(* IEC 61131-3 sources: Industry-PLC-LLM/data/PLCBEAD_repo/PLCBEAD_PLCEmbed-main/PLC-BEAD/Source/GEB/Network_TN_SEND_ROWS, 1 file *)

(* ---- TN_SEND_ROWS.ST ---- *)
TYPE
  oscat_IP_FIFO128_DATA  : ARRAY [1..128] OF BYTE;
  oscat_Mailbox  : ARRAY [1..16] OF BYTE;

  oscat_IP_FIFO_DATA :
  STRUCT
    X       : oscat_IP_FIFO128_DATA; (* IP_ID FIFO Speicher          *)
    Y       : oscat_IP_FIFO128_DATA; (* IP_ID Z�hler                 *)
    ID      : BYTE;                  (* h�chste vergabene id         *)
    MAX_ID  : BYTE;                  (* maximal Anmeldungen pro ID   *)
    INIT    : BOOL;                  (* Initialisierung durchgef�hrt *)
    EMPTY   : BOOL;                  (* FIFO leer                    *)
    FULL    : BOOL;                  (* FIFO voll                    *)
    TOP     : INT;                   (* maximale anzahl IN FIFO      *)
    NW      : INT;                   (* Schreibzeiger                *)
    NR      : INT;                   (* Lesezeiger                   *)
  END_STRUCT;

  oscat_IP_C:
  STRUCT
    C_MODE:			BYTE;          		(*W Mode: TCP/UCP AKTIV/PASSIV                               *)
    C_PORT:         WORD;          		(*W Portnummer                                               *)
    C_IP:           DWORD;         		(*W IP-ADRESSe gepackt wwxxyyzz = www.xxx.yyy.zzz            *)
    C_STATE:        BYTE;          		(*R VerbindungsSTATUS ON/OFF + Flanke ON/OFF                 *)
    C_ENABLE:       BOOL;          		(*W Freigabe f�r Connect                                     *)
    R_OBSERVE:      BOOL;          		(*W Empfang ueberwachen                                      *)
    TIME_RESET:     BOOL;          		(*W Alle Timer ruecksetzen                                   *)
    ERROR:          DWORD;         		(*R vvwwxxyy (vv = CON_ERROR, ww = SEN_ERROR, xx = REC_ERROR *)
    FIFO:           oscat_IP_FIFO_DATA; (*I IP FIFO Struktur                                         *)
    MAILBOX:		oscat_Mailbox;		(*I Mailbox: Datenbereich f�r Bausteindatenaustausch         *)
    END_STRUCT;
END_TYPE

TYPE

  oscat_NW_BUF_LONG  : ARRAY [0..4095] OF BYTE;

  oscat_NETWORK_BUFFER :
  STRUCT
    SIZE   : UINT;
    BUFFER : oscat_NW_BUF_LONG;
  END_STRUCT;

END_TYPE

TYPE

  bya_TN_CHAR:       	ARRAY [0..1919] OF BYTE;
  bya_TN_BACKUP:     	ARRAY [0..1919] OF BYTE;
  bya_TN_COLOR:      	ARRAY [0..1919] OF BYTE;
  bya_TN_Line_Update:	ARRAY [0..23]   OF BOOL;

  us_TN_SCREEN :
  STRUCT
    bya_CHAR:			bya_TN_CHAR;
    bya_COLOR:			bya_TN_COLOR;
    bya_BACKUP:			bya_TN_BACKUP;
    bya_Line_Update:	bya_TN_Line_Update;

    by_Input_Exten_Code:    BYTE;
    by_Input_ASCII_Code:    BYTE;
    bo_Input_ASCII_IsNum:   BOOL;
    in_Page_Number:        	INT;                (* aktive Seiten-Nr.              *)
    in_Cursor_X:           	INT;                (* Cursor X-POSition              *)
    in_Cursor_Y:           	INT;                (* Cursor Y-POSition              *)
    in_EOS_Offset:         	INT;                (* End of String Offset           *)
    by_Clear_Screen_Attr:  	BYTE;               (* Clear-Screen Attr              *)
    bo_Clear_Screen:       	BOOL;               (* Clear-Screen ausl�sen          *)
    bo_Modal_Dialog:       	BOOL;               (* Modaler Dialog ist aktiv       *)
    bo_Menue_Bar_Dialog:   	BOOL;               (* Menue Dialog ist aktiv         *)

  END_STRUCT;
END_TYPE

FUNCTION INT_TO_BCDC:BYTE

	VAR_INPUT
		IN :	INT;
	END_VAR

	INT_TO_BCDC := SHL(INT_TO_BYTE(IN / INT#10),4) OR INT_TO_BYTE(IN MOD INT#10);

END_FUNCTION

FUNCTION_BLOCK TN_SEND_ROWS_Block

  VAR_IN_OUT
    IP_C :	oscat_IP_C;
    S_BUF :	oscat_NETWORK_BUFFER;
    Xus_TN_SCREEN :	us_TN_SCREEN;
  END_VAR

  VAR_INPUT
    S_BUF_SIZE :	INT;
  END_VAR

  VAR
    in_Line_Count :	INT;
    in_Col_Count :	INT;
    in_Last_Row_Index :	INT;
    bo_Break_Loop :	BOOL;
    in_Row_Count :	INT;
    in_Offset :	INT;
    in_Write_Index :	INT;
    in_Write_Index_Backup :	INT;
    by_Cur_Color :	BYTE;
    by_last_Color :	BYTE;
    in_Write_STOP :	INT;
  END_VAR

  IF (IP_C.C_STATE < BYTE#127 OR S_BUF.SIZE > UINT#0) THEN
    RETURN;
  END_IF;

  in_Write_Index := UINT_TO_INT(S_BUF.SIZE) - 1;

  in_Write_Index_Backup := in_Write_Index;

  IF (IP_C.C_STATE = BYTE#254) OR (Xus_TN_SCREEN.bo_Clear_Screen) THEN

    Xus_TN_SCREEN.bo_Clear_Screen := FALSE;

    FOR in_Line_Count := INT#00 TO INT#23 DO
      Xus_TN_SCREEN.bya_Line_Update[in_Line_Count] := TRUE;
    END_FOR;

    in_Write_Index := in_Write_Index + INT#1;
    S_BUF.BUFFER[in_Write_Index] := BYTE#16#1B;
    in_Write_Index := in_Write_Index + INT#1;
    S_BUF.BUFFER[in_Write_Index] := BYTE#16#5B;
    in_Write_Index := in_Write_Index + INT#1;
    S_BUF.BUFFER[in_Write_Index] := BYTE#16#30;
    in_Write_Index := in_Write_Index + INT#1;
    S_BUF.BUFFER[in_Write_Index] := BYTE#16#3B;
    in_Write_Index := in_Write_Index + INT#1;
    S_BUF.BUFFER[in_Write_Index] := BYTE#16#33;

    in_Write_Index := in_Write_Index + INT#1;
    S_BUF.BUFFER[in_Write_Index] := (SHR(Xus_TN_SCREEN.by_Clear_Screen_Attr,4) OR BYTE#16#30);

    in_Write_Index := in_Write_Index + INT#1;
    S_BUF.BUFFER[in_Write_Index] := BYTE#16#3B;
    in_Write_Index := in_Write_Index + INT#1;
    S_BUF.BUFFER[in_Write_Index] := BYTE#16#34;

    in_Write_Index := in_Write_Index + INT#1;
    S_BUF.BUFFER[in_Write_Index] := ((Xus_TN_SCREEN.by_Clear_Screen_Attr AND BYTE#16#07) OR BYTE#16#30);

    in_Write_Index := in_Write_Index + INT#1;
    S_BUF.BUFFER[in_Write_Index] := BYTE#16#6D;

    in_Write_Index := in_Write_Index + INT#1;
    S_BUF.BUFFER[in_Write_Index] := BYTE#16#1B;
    in_Write_Index := in_Write_Index + INT#1;
    S_BUF.BUFFER[in_Write_Index] := BYTE#16#5B;
    in_Write_Index := in_Write_Index + INT#1;
    S_BUF.BUFFER[in_Write_Index] := BYTE#16#32;
    in_Write_Index := in_Write_Index + INT#1;
    S_BUF.BUFFER[in_Write_Index] := BYTE#16#4A;

    in_Write_Index := in_Write_Index + INT#1;
    S_BUF.BUFFER[in_Write_Index] := BYTE#16#1B;
    in_Write_Index := in_Write_Index + INT#1;
    S_BUF.BUFFER[in_Write_Index] := BYTE#16#5B;
    in_Write_Index := in_Write_Index + INT#1;
    S_BUF.BUFFER[in_Write_Index] := BYTE#16#3F;
    in_Write_Index := in_Write_Index + INT#1;
    S_BUF.BUFFER[in_Write_Index] := BYTE#16#37;
    in_Write_Index := in_Write_Index + INT#1;
    S_BUF.BUFFER[in_Write_Index] := BYTE#16#6C;

  END_IF;

  in_Last_Row_Index := INT#0;
  bo_Break_Loop := FALSE;
  in_Write_STOP := S_BUF_SIZE-20;

  FOR in_Line_Count := 0 TO 23 DO

    in_Offset := in_Row_Count * INT#80;

    IF (Xus_TN_SCREEN.bya_Line_Update[in_Row_Count] = TRUE) THEN

      in_Write_Index := in_Write_Index + INT#1;
      S_BUF.BUFFER[in_Write_Index] := BYTE#16#1B;
      in_Write_Index := in_Write_Index + INT#1;
      S_BUF.BUFFER[in_Write_Index] := BYTE#16#5B;

      in_Write_Index := in_Write_Index + INT#1;
      S_BUF.BUFFER[in_Write_Index] :=
        SHR(INT_TO_BCDC(in_Row_Count + INT#1),INT#4) OR BYTE#16#30;

      in_Write_Index := in_Write_Index + INT#1;
      S_BUF.BUFFER[in_Write_Index] :=
        (INT_TO_BCDC(in_Row_Count + INT#1) AND BYTE#16#0F) OR BYTE#16#30;

      in_Write_Index := in_Write_Index + INT#1;
      S_BUF.BUFFER[in_Write_Index] := BYTE#16#3B;
      in_Write_Index := in_Write_Index + INT#1;
      S_BUF.BUFFER[in_Write_Index] := BYTE#16#31;
      in_Write_Index := in_Write_Index + INT#1;
      S_BUF.BUFFER[in_Write_Index] := BYTE#16#48;

      FOR in_Col_Count := 0 TO 79 DO

        by_Cur_Color := Xus_TN_SCREEN.bya_COLOR[in_Offset];
        IF (by_Cur_Color <> by_last_Color) OR (in_Col_Count = INT#00) THEN

          in_Write_Index := in_Write_Index + INT#1;
          S_BUF.BUFFER[in_Write_Index] := BYTE#16#1B;

          in_Write_Index := in_Write_Index + INT#1;
          S_BUF.BUFFER[in_Write_Index] := BYTE#16#5B;

          IF  (((by_Cur_Color AND BYTE#2#10001000) XOR (by_last_Color AND BYTE#2#10001000)) <> BYTE#00) OR (in_Col_Count = 0) THEN

            in_Write_Index := in_Write_Index + INT#1;
            S_BUF.BUFFER[in_Write_Index] := BYTE#16#30;
            in_Write_Index := in_Write_Index + INT#1;
            S_BUF.BUFFER[in_Write_Index] := BYTE#16#3B;

            IF (by_Cur_Color AND BYTE#2#00001000) = BYTE#2#00000000 THEN

              in_Write_Index := in_Write_Index + INT#1;
              S_BUF.BUFFER[in_Write_Index] := BYTE#16#31;
              in_Write_Index := in_Write_Index + INT#1;
              S_BUF.BUFFER[in_Write_Index] := BYTE#16#3B;

            END_IF;

            IF (by_Cur_Color AND BYTE#2#10000000) = BYTE#2#10000000 THEN

              in_Write_Index := in_Write_Index + INT#1;
              S_BUF.BUFFER[in_Write_Index] := BYTE#16#35;
              in_Write_Index := in_Write_Index + INT#1;
              S_BUF.BUFFER[in_Write_Index] := BYTE#16#3B;

            END_IF;

          END_IF;

          in_Write_Index := in_Write_Index + INT#1;
          S_BUF.BUFFER[in_Write_Index] := BYTE#16#33;

          in_Write_Index := in_Write_Index + INT#1;
          S_BUF.BUFFER[in_Write_Index] := ((SHR(by_Cur_Color,4) AND BYTE#2#00000111) OR BYTE#16#30);

          in_Write_Index := in_Write_Index + INT#1;
          S_BUF.BUFFER[in_Write_Index] := BYTE#16#3B;

          in_Write_Index := in_Write_Index + INT#1;
          S_BUF.BUFFER[in_Write_Index] := BYTE#16#34;

          in_Write_Index := in_Write_Index + INT#1;
          S_BUF.BUFFER[in_Write_Index] := ((by_Cur_Color AND BYTE#2#00000111) OR BYTE#16#30);

          in_Write_Index := in_Write_Index + INT#1;
          S_BUF.BUFFER[in_Write_Index] := BYTE#16#6D;

          by_last_Color := by_Cur_Color;

        END_IF;

        IF (in_Write_Index > in_Write_STOP) THEN

          bo_Break_Loop := TRUE;
          EXIT;

        END_IF;

        in_Write_Index := in_Write_Index + INT#1;
        S_BUF.BUFFER[in_Write_Index] := Xus_TN_SCREEN.bya_CHAR[in_Offset];

        in_Offset := in_Offset + INT#01;
      END_FOR;

      IF (bo_Break_Loop = TRUE) THEN

        in_Write_Index := in_Last_Row_Index;

        EXIT;
      END_IF;

      in_Last_Row_Index := in_Write_Index;
      Xus_TN_SCREEN.bya_Line_Update[in_Row_Count] := FALSE;

    END_IF;

    in_Row_Count := in_Row_Count + INT#01;

    IF (in_Row_Count > INT#23) THEN
      in_Row_Count := INT#00;
    END_IF;

  END_FOR;

  IF (bo_Break_Loop = FALSE) THEN

    in_Row_Count := INT#00;

  END_IF;

  IF (in_Write_Index <> in_Write_Index_Backup) THEN

    in_Write_Index := in_Write_Index + INT#1;
    S_BUF.BUFFER[in_Write_Index] := BYTE#16#1B;
    in_Write_Index := in_Write_Index + INT#1;
    S_BUF.BUFFER[in_Write_Index] := BYTE#16#5B;

    in_Write_Index := in_Write_Index + INT#1;
    S_BUF.BUFFER[in_Write_Index] := SHR(INT_TO_BCDC(Xus_TN_SCREEN.in_Cursor_Y + 1),INT#4) OR BYTE#16#30;

    in_Write_Index := in_Write_Index + INT#1;
    S_BUF.BUFFER[in_Write_Index] := (INT_TO_BCDC(Xus_TN_SCREEN.in_Cursor_Y + 1) AND BYTE#16#0F) OR BYTE#16#30;

    in_Write_Index := in_Write_Index + INT#1;
    S_BUF.BUFFER[in_Write_Index] := BYTE#16#3B;

    in_Write_Index := in_Write_Index + INT#1;
    S_BUF.BUFFER[in_Write_Index] := SHR(INT_TO_BCDC(Xus_TN_SCREEN.in_Cursor_X + 1),INT#4) OR BYTE#16#30;

    in_Write_Index := in_Write_Index + INT#1;
    S_BUF.BUFFER[in_Write_Index] := (INT_TO_BCDC(Xus_TN_SCREEN.in_Cursor_X + 1) AND BYTE#16#0F) OR BYTE#16#30;

    in_Write_Index := in_Write_Index + INT#1;
    S_BUF.BUFFER[in_Write_Index] := BYTE#16#48;

  END_IF;

  S_BUF.SIZE := INT_TO_UINT(in_Write_Index + 1);

END_FUNCTION_BLOCK

PROGRAM program0
	VAR
		IP_C :	oscat_IP_C;
    S_BUF :	oscat_NETWORK_BUFFER;
    Xus_TN_SCREEN :	us_TN_SCREEN;
    S_BUF_SIZE :	INT;

		func_block : TN_SEND_ROWS_Block;
	END_VAR
	func_block.IP_C := IP_C;
  func_block.S_BUF := S_BUF;
  func_block.Xus_TN_SCREEN := Xus_TN_SCREEN;
  func_block.S_BUF_SIZE := S_BUF_SIZE;

	func_block();
	IP_C  := func_block.IP_C;
  S_BUF  := func_block.S_BUF;
  Xus_TN_SCREEN  := func_block.Xus_TN_SCREEN;
END_PROGRAM
